Fanuc KAREL source: kc00019.KL

-- PROVISIONAL review KL for V770-1; original PC SHA256 f5cebec8397a8f1fb12013ac5494f2d5d227d116d3eb51c32df800948bd7353d
-- Incomplete behavior may be omitted. Consult companion uncertainty JSON. Do not deploy.
PROGRAM KC00019
%NOLOCKGROUP
BEGIN
  -- UNRESOLVED_PC offsets 5-53; opcodes 27,22,22,22,22,22,2A,22,22,31
  -- UNRESOLVED_PC offsets 58-62; opcodes 7F
END KC00019
